TYPE ST_LAST_STEPS :
STRUCT
	strStepName: 		    STRING;
	iStepID:			      INT;
	tStepTime: 			    TIME;
	tDelayTime:			    TIME;
	eStepType:			    BOOL;
	bBreakpointActive: 	BOOL;
	bDisableBreakpoint: BOOL;
END_STRUCT
END_TYPE

(* stored: Version 1.1.0.1, ProductVersion 3.1.4024.12
   DUT ST_LAST_STEPS: Id {abbf059d-d576-47af-a510-47b14f3ddea4} *)
